TYPE ObjectId_t : STRING; END_TYPE

(* stored: Version 1.1.0.1, ProductVersion 3.1.4022.12
   DUT ObjectId_t: Id {ec3254fd-e180-4792-8396-8a521f2cea29} *)
